// This function has been automatically generated from the project information.
VAR_GLOBAL CONSTANT
	{attribute 'const_non_replaced'}
	stLibVersion_BasePpt : ST_LibVersion := (iMajor := 0, iMinor := 0, iBuild := 0, iRevision := 51, sVersion := '0.0.0.51');
END_VAR

(* stored: Version 1.1.0.1, ProductVersion 3.1.0.26
   GVL Global_Version: Id {e072c35e-68b4-43ec-9139-5f2ac659c52b} *)
